(* CODESYS project codesys_code_execution_speedTests.export
   Author: Toni Kucic
   Version: 1.0
   Description: Cheatsheet for programming a PLC in IEC61131-3 Structured text. Contains usage of operators and common functions.
   Title: Plc Structured Text Cheatsheet
   CompiledLibraryCompatibilityVersion: CODESYS V3.5 SP16
   Company: TK Automation

Project tree, tasks and I/O mapping:
  CODESYS_Control_Win_V3_x64 : CODESYS Control Win V3 x64, 3S - Smart Software Solutions GmbH, version 3.5.18.20
    application Application
      libraries: MemoryUtils, 3.5.18.0 (3S - Smart Software Solutions GmbH)
      task Task (cyclic, interval 200 ms, priority 1) calls speedRunner
  CODESYS_Control_RTE_V3_x64 : CODESYS Control RTE V3 x64, 3S - Smart Software Solutions GmbH, version 3.5.18.20
    application Application
      libraries: MemoryUtils, 3.5.18.0 (3S - Smart Software Solutions GmbH)
      task Task (cyclic, interval 200 ms, priority 1) calls speedRunner
  libraries: Standard, 3.5.18.0 (System)
  01 - Impact of dynamic arrays/
    program x01_ImpactOfDynamicArrays [ST]
  02 - Execution speed of PLC languages/
    program x02_ExecSpeedOfLanguageTypes [ST]
    function addTwoIntsLadder [LD]
    function addTwoIntsST [ST]
    function addTwoIntsFBD [FBD]
  03 - Floating point operations/
    program x03_FloatingPointOperations [ST]
  04 - Function overhead/
    function addTwoInts [ST]
    program x04_FunctionOverhead [ST]: addTwoNumbers
  05 - MemSet over Data Zero/
    program x05_MemSetVsDataZeero [ST]
    data type dtTestStruct
  06 - SHL over MemCpy/
    program x06_ShlVsMemCpy [ST]
  07 - String operations/
    program x07_StringOperations [ST]
  08 - Operations with booleans/
    program x08_CheckingBools [ST]
  09 - Case versus IF ELSIF/
    program x09_CaseVsIfElsif [ST]: returnIndexIfElsif, returnIndexCase
  10 - Bit operations/
    program x10_1_BitAccess [ST]
    data type dtBitStruct
    program x10_3_BitMath [ST]
    program x10_2_BitSet [ST]
    function checkBit_bitmask [ST]
    function setBit_bitmask [ST]
    function clearBit_bitmask [ST]
    function setBitToValue_bitmask [ST]
    function setBit_dotNot [ST]
    function checkBit_dotNot [ST]
    function clearBit_dotNot [ST]
    function checkBit_bitStruct [ST]
    function clearBit_bitStruct [ST]
    function setBit_bitStruct [ST]
    function setBitToValue_bitStruct [ST]
    function setBitToValue_dotNot [ST]
  TestFramework/
    function calcAVG [ST]
    data type dtSpeedTest
    program speedRunner [ST]
*)

// 05 - MemSet over Data Zero/dtTestStruct
TYPE dtTestStruct :
STRUCT
	dummy1 : USINT := 255;
	Elem1 : INT := -1;
	Id : DWORD := 215215126;
	IdText : STRING := 'Testing for speed';
	dummy2 : ARRAY[0..11] OF DWORD;
	dummy4 : BOOL := FALSE;
	dummy5 : STRING[255] := 'Big array';
	dummy6 : LINT := 1211212723838939;
END_STRUCT
END_TYPE

// 10 - Bit operations/dtBitStruct
TYPE dtBitStruct :
STRUCT
	bit1 : BIT;
	bit2 : BIT;
	bit3 : BIT;
	bit4 : BIT;
	bit5 : BIT;
	bit6 : BIT;
	bit7 : BIT;
	bit8 : BIT;
	bit9 : BIT;
	bit10 : BIT;
	bit11 : BIT;
	bit12 : BIT;
	bit13 : BIT;
	bit14 : BIT;
	bit15 : BIT;
	bit16 : BIT;
END_STRUCT
END_TYPE

// TestFramework/dtSpeedTest
TYPE dtSpeedTest :
STRUCT
	Results 			: ARRAY[0..9] OF LTIME;
	AverageExecTime  	: LTIME;
	OldTime     		: LTIME;
	ExecTime    		: LTIME;
END_STRUCT
END_TYPE

// TestFramework/speedRunner
PROGRAM speedRunner
VAR
	vOldTime : LTIME;
	vTimeToRunTests : LTIME;
	vStart : BOOL := TRUE;
END_VAR

IF vStart THEN
	vOldTime := LTIME();
	vStart := FALSE;
END_IF

(*Run tests one by one*)
x01_ImpactOfDynamicArrays();
x02_ExecSpeedOfLanguageTypes();
x03_FloatingPointOperations();
x04_FunctionOverhead();
x05_MemSetVsDataZeero();
x06_ShlVsMemCpy();
x07_StringOperations();
x08_CheckingBools();
x09_CaseVsIfElsif();
x10_1_BitAccess();
x10_2_BitSet();
x10_3_BitMath();

IF x01_ImpactOfDynamicArrays.vRunDone
AND x02_ExecSpeedOfLanguageTypes.vRunDone
AND x03_FloatingPointOperations.vRunDone
AND x04_FunctionOverhead.vRunDone
AND x05_MemSetVsDataZeero.vRunDone
AND x06_ShlVsMemCpy.vRunDone
AND x07_StringOperations.vRunDone
AND x08_CheckingBools.vRunDone
AND x09_CaseVsIfElsif.vRunDone
AND x10_1_BitAccess.vRunDone
AND x10_2_BitSet.vRunDone
AND x10_3_BitMath.vRunDone
AND vTimeToRunTests = LTIME#0S
 THEN
	vTimeToRunTests := LTIME() - vOldTime;
END_IF

END_PROGRAM

// 01 - Impact of dynamic arrays/x01_ImpactOfDynamicArrays
PROGRAM x01_ImpactOfDynamicArrays
VAR CONSTANT
	cNrRuns : USINT(0..9) := 5;
	cRepeatCalcTimes : UDINT := 1000000; //1 Million times
END_VAR
VAR
	vRunsCompleted : USINT := 0;
	vRunDone : BOOL := FALSE;
	vTest1 : dtSpeedTest;
	vTest2 : dtSpeedTest;

	i : UDINT;
	
	//Test vars
	vAvgTimeFun : LTIME;
	vAvgTimeHardCoded : LTIME;
	vTimes : ARRAY[0..9] OF LTIME := [LTIME#1MS,LTIME#2MS,LTIME#3MS,LTIME#4MS,LTIME#5MS,LTIME#6MS,LTIME#7MS,LTIME#8MS,LTIME#9MS,LTIME#10MS];
	j : USINT;
END_VAR

IF vRunsCompleted > cNrRuns THEN
	vTest1.AverageExecTime := calcAvg(vTest1.Results);
	vTest2.AverageExecTime := calcAvg(vTest2.Results);
	vRunDone := TRUE;
	RETURN;
END_IF
	
//------------CALCULATION A -------------------
vTest1.OldTime := LTIME();
FOR i:= 0 TO cRepeatCalcTimes DO
	vAvgTimeFun := calcAvg(vTimes);
END_FOR
vTest1.ExecTime := LTIME() - vTest1.OldTime;

//------------CALCULATION B -------------------
vTest2.OldTime := LTIME();
FOR i:= 0 TO cRepeatCalcTimes DO
	vAvgTimeHardCoded := LTIME#0MS;
	FOR j:= 0 TO 9 DO
		vAvgTimeHardCoded := vAvgTimeHardCoded + vTimes[j];
	END_FOR
	vAvgTimeHardCoded := vAvgTimeHardCoded / j;
END_FOR
vTest2.ExecTime := LTIME() - vTest2.OldTime;

//------------CATCH RESULTS---------------------
vTest1.Results[vRunsCompleted] := vTest1.ExecTime;
vTest2.Results[vRunsCompleted] := vTest2.ExecTime;
vRunsCompleted := vRunsCompleted + 1;

END_PROGRAM

// TestFramework/calcAVG
FUNCTION calcAVG : LTIME
VAR_IN_OUT
	Results : ARRAY[*] OF LTIME;
END_VAR
VAR
	i : DINT;
END_VAR

FOR i:= LOWER_BOUND(Results,1) TO UPPER_BOUND(Results,1) DO
	calcAvg := calcAvg + Results[i];
END_FOR
calcAvg := calcAvg / i;
RETURN;

END_FUNCTION

// 02 - Execution speed of PLC languages/x02_ExecSpeedOfLanguageTypes
PROGRAM x02_ExecSpeedOfLanguageTypes
VAR CONSTANT
	cNrRuns : USINT(0..9) := 5;
	cRepeatCalcTimes : UDINT := 1000000; //1 Million times
END_VAR
VAR
	vRunsCompleted : USINT := 0;
	vRunDone : BOOL := FALSE;
	vTest1 : dtSpeedTest;
	vTest2 : dtSpeedTest;
	vTest3 : dtSpeedTest;
	i : UDINT;
	
	//Test vars
	vInt1 : INT := 1;
	vInt2 : INT := 2;
	vResult1 : INT;
	vResult2 : INT;
	vResult3 : INT;
END_VAR

IF vRunsCompleted > cNrRuns THEN
	vTest1.AverageExecTime := calcAvg(vTest1.Results); //User function Ladder
	vTest2.AverageExecTime := calcAvg(vTest2.Results); //User function ST
	vTest3.AverageExecTime := calcAvg(vTest3.Results); //User function FBD
	vRunDone := TRUE;
	RETURN;
END_IF
	
//------------CALCULATION A -------------------
vTest1.OldTime := LTIME();
FOR i:= 0 TO cRepeatCalcTimes DO
	vResult1 := addTwoIntsLadder(vInt1, vInt2);
END_FOR
vTest1.ExecTime := LTIME() - vTest1.OldTime;

//------------CALCULATION B -------------------
vTest2.OldTime := LTIME();
FOR i:= 0 TO cRepeatCalcTimes DO
	vResult2 := addTwoIntsST(vInt1, vInt2);
END_FOR
vTest2.ExecTime := LTIME() - vTest2.OldTime;

//------------CALCULATION C -------------------
vTest3.OldTime := LTIME();
FOR i:= 0 TO cRepeatCalcTimes DO
	vResult3 := addTwoIntsFBD(vInt1, vInt2);
END_FOR
vTest3.ExecTime := LTIME() - vTest3.OldTime;

//------------CATCH RESULTS---------------------
vTest1.Results[vRunsCompleted] := vTest1.ExecTime;
vTest2.Results[vRunsCompleted] := vTest2.ExecTime;
vTest3.Results[vRunsCompleted] := vTest3.ExecTime;
vRunsCompleted := vRunsCompleted + 1;

END_PROGRAM

// 02 - Execution speed of PLC languages/addTwoIntsLadder
FUNCTION addTwoIntsLadder : INT
VAR_INPUT
	Int1 : INT;
	Int2 : INT;
END_VAR
VAR
END_VAR

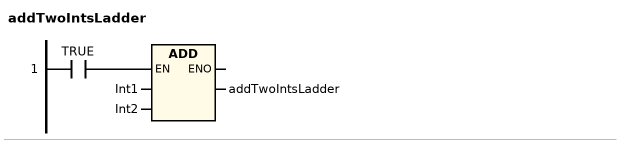
// NETWORK 1
addTwoIntsLadder := Int1 + Int2;

END_FUNCTION

// 02 - Execution speed of PLC languages/addTwoIntsST
FUNCTION addTwoIntsST : INT
VAR_INPUT
	int1 : INT;
	int2 : INT;
END_VAR
VAR
END_VAR

addTwoIntsST := int1 + int2;

END_FUNCTION

// 02 - Execution speed of PLC languages/addTwoIntsFBD
FUNCTION addTwoIntsFBD : INT
VAR_INPUT
	int1 : INT;
	int2 : INT;
END_VAR
VAR
END_VAR

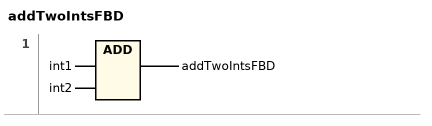
// NETWORK 1
addTwoIntsFBD := int1 + int2;

END_FUNCTION

// 03 - Floating point operations/x03_FloatingPointOperations
PROGRAM x03_FloatingPointOperations
VAR CONSTANT
	cNrRuns : USINT(0..9) := 5;
	cRepeatCalcTimes : UDINT := 1000000; //1 Million times
END_VAR
VAR
	vRunsCompleted : USINT := 0;
	vRunDone : BOOL := FALSE;
	vTest1 : dtSpeedTest;
	vTest2 : dtSpeedTest;
	vTest3 : dtSpeedTest;
	vTest4 : dtSpeedTest;
	vTest5 : dtSpeedTest;
	vTest6 : dtSpeedTest;
	vTest7 : dtSpeedTest;
	vTest8 : dtSpeedTest;
	vTest9 : dtSpeedTest;
	i : UDINT;
	
	//Test vars
	vInteger1 : INT := 1234;
	vInteger2 : INT := 4231;
	vReal1 : REAL := 1234.4231;
	vReal2 : REAL := 4231.1234;
	vInteger3 : DINT := 1234;
	vInteger4 : DINT := 4231;
	
	vResult1 : INT;
	vResult2 : REAL;
	vResult3 : DINT;
	vResult4 : INT;
	vResult5 : REAL;
	vResult6 : DINT;
	vResult7 : INT;
	vResult8 : REAL;
	vResult9 : DINT;
END_VAR

IF vRunsCompleted > cNrRuns THEN
	vTest1.AverageExecTime := calcAvg(vTest1.Results); //Time to add two integers 1 milion times
	vTest2.AverageExecTime := calcAvg(vTest2.Results); //Time to add two reals 1 milion times
	vTest3.AverageExecTime := calcAvg(vTest3.Results); //Time to add two DINTs (32b INT) 1 milion times
	vTest4.AverageExecTime := calcAvg(vTest4.Results); //Time to multiply two integers 1 milion times
	vTest5.AverageExecTime := calcAvg(vTest5.Results); //Time to multiply two reals 1 milion times
	vTest6.AverageExecTime := calcAvg(vTest6.Results); //Time to multiply two DINTs (32b INT) 1 milion times
	vTest7.AverageExecTime := calcAvg(vTest7.Results); //Time to divide two integers 1 milion times
	vTest8.AverageExecTime := calcAvg(vTest8.Results); //Time to divide two reals 1 milion times
	vTest9.AverageExecTime := calcAvg(vTest9.Results); //Time to divide two DINTs (32b INT) 1 milion times
	vRunDone := TRUE;	
	RETURN;
END_IF

//------------CALCULATION A -------------------
vTest1.OldTime := LTIME();
FOR i:= 0 TO cRepeatCalcTimes DO
	vResult1 := vInteger1 + vInteger2;
END_FOR
vTest1.ExecTime := LTIME() - vTest1.OldTime;

//------------CALCULATION B -------------------
vTest2.OldTime := LTIME();
FOR i:= 0 TO cRepeatCalcTimes DO
	vResult2 := vReal1 + vReal2;
END_FOR
vTest2.ExecTime := LTIME() - vTest2.OldTime;

//------------CALCULATION C -------------------
vTest3.OldTime := LTIME();
FOR i:= 0 TO cRepeatCalcTimes DO
	vResult3 := vInteger3 + vInteger4;
END_FOR
vTest3.ExecTime := LTIME() - vTest3.OldTime;

//------------CALCULATION D -------------------
vTest4.OldTime := LTIME();
FOR i:= 0 TO cRepeatCalcTimes DO
	vResult4 := vInteger1 * vInteger2;
END_FOR
vTest4.ExecTime := LTIME() - vTest4.OldTime;

//------------CALCULATION E -------------------
vTest5.OldTime := LTIME();
FOR i:= 0 TO cRepeatCalcTimes DO
	vResult5 := vReal1 * vReal2;
END_FOR
vTest5.ExecTime := LTIME() - vTest5.OldTime;

//------------CALCULATION F -------------------
vTest6.OldTime := LTIME();
FOR i:= 0 TO cRepeatCalcTimes DO
	vResult6 := vInteger3 * vInteger4;
END_FOR
vTest6.ExecTime := LTIME() - vTest6.OldTime;

//------------CALCULATION G -------------------
vTest7.OldTime := LTIME();
FOR i:= 0 TO cRepeatCalcTimes DO
	vResult7 := vInteger1 / vInteger2;
END_FOR
vTest7.ExecTime := LTIME() - vTest7.OldTime;

//------------CALCULATION H -------------------
vTest8.OldTime := LTIME();
FOR i:= 0 TO cRepeatCalcTimes DO
	vResult8 := vReal1 / vReal2;
END_FOR
vTest8.ExecTime := LTIME() - vTest8.OldTime;

//------------CALCULATION I -------------------
vTest9.OldTime := LTIME();
FOR i:= 0 TO cRepeatCalcTimes DO
	vResult9 := vInteger3 / vInteger4;
END_FOR
vTest9.ExecTime := LTIME() - vTest9.OldTime;


//------------CATCH RESULTS---------------------
vTest1.Results[vRunsCompleted] := vTest1.ExecTime;
vTest2.Results[vRunsCompleted] := vTest2.ExecTime;
vTest3.Results[vRunsCompleted] := vTest3.ExecTime;
vTest4.Results[vRunsCompleted] := vTest4.ExecTime;
vTest5.Results[vRunsCompleted] := vTest5.ExecTime;
vTest6.Results[vRunsCompleted] := vTest6.ExecTime;
vTest7.Results[vRunsCompleted] := vTest7.ExecTime;
vTest8.Results[vRunsCompleted] := vTest8.ExecTime;
vTest9.Results[vRunsCompleted] := vTest9.ExecTime;
vRunsCompleted := vRunsCompleted + 1;

END_PROGRAM

// 04 - Function overhead/x04_FunctionOverhead
PROGRAM x04_FunctionOverhead
VAR CONSTANT
	cNrRuns : USINT(0..9) := 5;
	cRepeatCalcTimes : UDINT := 1000000; //1 Million times
END_VAR
VAR
	vRunsCompleted : USINT := 0;
	vRunDone : BOOL := FALSE;
	vTest1 : dtSpeedTest;
	vTest2 : dtSpeedTest;
	vTest3 : dtSpeedTest;

	i : UDINT;
	
	//Test vars
	vInt1 : INT := 1;
	vInt2 : INT := 2;
	vResult1 : INT;
	vResult2 : INT;
	vResult3 : INT;
END_VAR

IF vRunsCompleted > cNrRuns THEN
	vTest1.AverageExecTime := calcAvg(vTest1.Results); //Operands
	vTest2.AverageExecTime := calcAvg(vTest2.Results); //User function
	vTest3.AverageExecTime := calcAvg(vTest3.Results); //PRG method
	vRunDone := TRUE;
	RETURN;
END_IF
	
//------------CALCULATION A -------------------
vTest1.OldTime := LTIME();
FOR i:= 0 TO cRepeatCalcTimes DO
	vResult1 := vInt1 + vInt2;
END_FOR
vTest1.ExecTime := LTIME() - vTest1.OldTime;

//------------CALCULATION B -------------------
vTest2.OldTime := LTIME();
FOR i:= 0 TO cRepeatCalcTimes DO
	vResult2 := addTwoInts(vInt1, vInt2);
END_FOR
vTest2.ExecTime := LTIME() - vTest2.OldTime;

//------------CALCULATION C -------------------
vTest3.OldTime := LTIME();
FOR i:= 0 TO cRepeatCalcTimes DO
	vResult3 := addTwoNumbers(vInt1, vInt2);
END_FOR
vTest3.ExecTime := LTIME() - vTest3.OldTime;

//------------CATCH RESULTS---------------------
vTest1.Results[vRunsCompleted] := vTest1.ExecTime;
vTest2.Results[vRunsCompleted] := vTest2.ExecTime;
vTest3.Results[vRunsCompleted] := vTest3.ExecTime;
vRunsCompleted := vRunsCompleted + 1;

METHOD PUBLIC addTwoNumbers : INT
VAR_INPUT
	int1 : INT;
	int2 : INT;
END_VAR
addTwoNumbers := int1 + int2;
END_METHOD

END_PROGRAM

// 04 - Function overhead/addTwoInts
FUNCTION addTwoInts : INT
VAR_IN_OUT
	int1 : INT;
	int2 : INT;
END_VAR
VAR
END_VAR

addTwoInts := int1 + int2;

END_FUNCTION

// 05 - MemSet over Data Zero/x05_MemSetVsDataZeero
PROGRAM x05_MemSetVsDataZeero
VAR CONSTANT
	cNrRuns : USINT(0..9) := 5;
	cRepeatCalcTimes : UDINT := 1000000; //1 Million times
	cEmptyStruct : dtTestStruct;
END_VAR
VAR
	vRunsCompleted : USINT := 0;
	vRunDone : BOOL := FALSE;
	vTest1 : dtSpeedTest;
	vTest2 : dtSpeedTest;

	i : UDINT;
	
	//Test variables
	vResultStruct1 : dtTestStruct;
	vResultStruct2 : dtTestStruct;
END_VAR

IF vRunsCompleted > cNrRuns THEN
	vTest1.AverageExecTime := calcAvg(vTest1.Results);
	vTest2.AverageExecTime := calcAvg(vTest2.Results);
	vRunDone := TRUE;
	RETURN;
END_IF
	
//------------CALCULATION A -------------------
vTest1.OldTime := LTIME();
FOR i:= 0 TO cRepeatCalcTimes DO
	//RESET STRUCT WITH A EMPTY STRUCT
	vResultStruct1 := cEmptyStruct;
END_FOR
vTest1.ExecTime := LTIME() - vTest1.OldTime;

//------------CALCULATION B -------------------
vTest2.OldTime := LTIME();
FOR i:= 0 TO cRepeatCalcTimes DO
	//RESET STRUCT WITH MEM SET
	MEMUtils.MemSet(pbyBuffer:= ADR(vResultStruct2), byValue:= 16#0 , dwSize:= SIZEOF(vResultStruct2));
END_FOR
vTest2.ExecTime := LTIME() - vTest2.OldTime;

//------------CATCH RESULTS---------------------
vTest1.Results[vRunsCompleted] := vTest1.ExecTime;
vTest2.Results[vRunsCompleted] := vTest2.ExecTime;
vRunsCompleted := vRunsCompleted + 1;

END_PROGRAM

// 06 - SHL over MemCpy/x06_ShlVsMemCpy
PROGRAM x06_ShlVsMemCpy
VAR CONSTANT
	cNrRuns : USINT(0..9) := 5;
	cRepeatCalcTimes : UDINT := 1000000; //1 Million times
END_VAR
VAR
	vRunsCompleted : USINT := 0;
	vRunDone : BOOL := FALSE;
	vTest1 : dtSpeedTest;
	vTest2 : dtSpeedTest;

	i : UDINT;
	
	//Test vars
	vSHRInteger : UINT;
	vMcpyInteger : UINT;
	vBuffer : ARRAY[0..1] OF USINT := [16#55, 16#AA];
	
	vSHLOldTime : LTIME;
	vMcpyOldTime : LTIME;
	
	vSHLExecTime : LTIME;
	vMcpyExecTime : LTIME;
	
END_VAR

IF vRunsCompleted > cNrRuns THEN
	vTest1.AverageExecTime := calcAvg(vTest1.Results);
	vTest2.AverageExecTime := calcAvg(vTest2.Results);
	vRunDone := TRUE;
	RETURN;
END_IF
	

vTest1.OldTime := LTIME();
FOR i:= 0 TO cRepeatCalcTimes DO
	//Assemble an UINT from two USINTs using SHR operator
	vSHRInteger := vBuffer[0] + SHL(vBuffer[1],8);
END_FOR
vTest1.ExecTime := LTIME() - vTest1.OldTime;

vTest2.OldTime := LTIME();
FOR i:= 0 TO cRepeatCalcTimes DO
	//Assemble an UINT from two USINTs using MemCpy
	MEMUtils.MemCpy(pbyDest:= ADR(vMcpyInteger), pbySrc:= ADR(vBuffer) , dwSize:= SIZEOF(vMcpyInteger));
END_FOR
vTest2.ExecTime := LTIME() - vTest2.OldTime;

//Results
vTest1.Results[vRunsCompleted] := vTest1.ExecTime;
vTest2.Results[vRunsCompleted] := vTest2.ExecTime;
vRunsCompleted := vRunsCompleted + 1;

END_PROGRAM

// 07 - String operations/x07_StringOperations
PROGRAM x07_StringOperations
VAR CONSTANT
	cNrRuns : USINT(0..9) := 5;
	cRepeatCalcTimes : UDINT := 1000000; //1 Million times
END_VAR
VAR
	vRunsCompleted : USINT := 0;
	vRunDone : BOOL := FALSE;
	vTest1 : dtSpeedTest;
	vTest2 : dtSpeedTest;
	vTest3 : dtSpeedTest;
	vTest4 : dtSpeedTest;
	vTest5 : dtSpeedTest;
	vTest6 : dtSpeedTest;
	i : UDINT;
	
	//Test vars
	vString1 : STRING[255] := 'Test string1';
	vString2 : STRING := 'Test string2';
	vString3 : STRING := 'a';
	vString4 : STRING := 'a';
	vByte :	BYTE := 16#FF;
	vArrByte :	ARRAY[0..255] OF BYTE;
	vResult1 : STRING[255];
	vResult2 : STRING;
	vResult3 : STRING;
	vResult4 : STRING[255];
	vResult5 : BYTE;
	vResult6 : ARRAY[0..255] OF BYTE;
	vSizes : ARRAY[0..3] OF UDINT;
END_VAR

IF vRunsCompleted > cNrRuns THEN
	vTest1.AverageExecTime := calcAvg(vTest1.Results); //Time to copy a string[255] 1 Million times
	vTest2.AverageExecTime := calcAvg(vTest2.Results); //Time to copy a string 1 Million times
	vTest3.AverageExecTime := calcAvg(vTest3.Results); //Time to concatenate 1 Million times characters with STRING
	vTest4.AverageExecTime := calcAvg(vTest4.Results); //Time to concatenate 1 Million times  characters with STRING[255]
	vTest5.AverageExecTime := calcAvg(vTest5.Results); //Time to move a byte 1 Million times
	vTest6.AverageExecTime := calcAvg(vTest6.Results); //Time to copy an array of 255 BYTE 1 Million times
	vRunDone := TRUE;
	RETURN;
END_IF

vSizes[0] := SIZEOF(vString1); //Size is 255 characters + zero char
vSizes[1] := SIZEOF(vString2); //Size is 80 characters + zero char, default if no size specified
vSizes[2] := SIZEOF(vResult3); //Size is 81, even though we concatenated 1 Million characters. The rest were chopped off
vSizes[3] := SIZEOF(vResult4); //Size is expected 256, other 744 characters chopped off

//------------CALCULATION A -------------------
vTest1.OldTime := LTIME();
FOR i:= 0 TO cRepeatCalcTimes DO
	vResult1 := vString1;
END_FOR
vTest1.ExecTime := LTIME() - vTest1.OldTime;

//------------CALCULATION B -------------------
vTest2.OldTime := LTIME();
FOR i:= 0 TO cRepeatCalcTimes DO
	vResult2 := vString2;
END_FOR
vTest2.ExecTime := LTIME() - vTest2.OldTime;

//------------CALCULATION C -------------------
vTest3.OldTime := LTIME();
FOR i:= 0 TO cRepeatCalcTimes DO
	vResult3 := CONCAT(vResult3, vString3);
END_FOR
vTest3.ExecTime := LTIME() - vTest3.OldTime;

//------------CALCULATION D -------------------
vTest4.OldTime := LTIME();
FOR i:= 0 TO cRepeatCalcTimes DO
	vResult4 := CONCAT(vResult4, vString4);
END_FOR
vTest4.ExecTime := LTIME() - vTest4.OldTime;

//------------CALCULATION E -------------------
vTest5.OldTime := LTIME();
FOR i:= 0 TO cRepeatCalcTimes DO
	vResult5 := vByte;
END_FOR
vTest5.ExecTime := LTIME() - vTest5.OldTime;

//------------CALCULATION F -------------------
vTest6.OldTime := LTIME();
FOR i:= 0 TO cRepeatCalcTimes DO
	vResult6 := vArrByte;
END_FOR
vTest6.ExecTime := LTIME() - vTest6.OldTime;

//------------CATCH RESULTS---------------------
vTest1.Results[vRunsCompleted] := vTest1.ExecTime;
vTest2.Results[vRunsCompleted] := vTest2.ExecTime;
vTest3.Results[vRunsCompleted] := vTest3.ExecTime;
vTest4.Results[vRunsCompleted] := vTest4.ExecTime;
vTest5.Results[vRunsCompleted] := vTest5.ExecTime;
vTest6.Results[vRunsCompleted] := vTest6.ExecTime;
vRunsCompleted := vRunsCompleted + 1;

END_PROGRAM

// 08 - Operations with booleans/x08_CheckingBools
PROGRAM x08_CheckingBools
VAR CONSTANT
	cNrRuns : USINT(0..9) := 5;
	cRepeatCalcTimes : UDINT := 1000000; //1 Million times
END_VAR
VAR
	vRunsCompleted : USINT := 0;
	vRunDone : BOOL := FALSE;
	vTest1 : dtSpeedTest;
	vTest2 : dtSpeedTest;
	vTest3 : dtSpeedTest;
	vTest4 : dtSpeedTest;
	vTest5 : dtSpeedTest;
	i : UDINT;
	
	//Test vars
	vBool : BOOL := TRUE;
	vResult : BOOL;
	vCounter : UINT := 0;
	vCastedUint : UINT;
END_VAR

IF vRunsCompleted > cNrRuns THEN
	vTest1.AverageExecTime := calcAvg(vTest1.Results); //Time to run IF vBool = TRUE THEN 1 Million times
	vTest2.AverageExecTime := calcAvg(vTest2.Results); //Time to run IF vBool THEN 1 Million times
	vTest3.AverageExecTime := calcAvg(vTest3.Results); //Time to increment a counter using if sentence 1 Million times
	vTest4.AverageExecTime := calcAvg(vTest4.Results); //Time to increment a counter using bool to UINT 1 Million times
	vTest5.AverageExecTime := calcAvg(vTest5.Results); //Time to cast a bool to UINT 1 Million times
	vRunDone := TRUE;
	RETURN;
END_IF

//------------CALCULATION A -------------------
vTest1.OldTime := LTIME();
//FOR i:= 0 TO cRepeatCalcTimes DO
	IF vBool = TRUE THEN
		vResult := vBool;
	END_IF
//END_FOR
vTest1.ExecTime := LTIME() - vTest1.OldTime;

//------------CALCULATION B -------------------
vTest2.OldTime := LTIME();
//FOR i:= 0 TO cRepeatCalcTimes DO
	IF vBool THEN
		vResult := vBool;
	END_IF
//END_FOR
vTest2.ExecTime := LTIME() - vTest2.OldTime;

//------------CALCULATION C -------------------
vTest3.OldTime := LTIME();
//FOR i:= 0 TO cRepeatCalcTimes DO
	IF vBool THEN
		vCounter := vCounter + 1;
	END_IF
//END_FOR
vTest3.ExecTime := LTIME() - vTest3.OldTime;

//------------CALCULATION D -------------------
vTest4.OldTime := LTIME();
//FOR i:= 0 TO cRepeatCalcTimes DO
	vCounter := vCounter + BOOL_TO_UINT(vBool);
//END_FOR
vTest4.ExecTime := LTIME() - vTest4.OldTime;

//------------CALCULATION D -------------------
vTest5.OldTime := LTIME();
//FOR i:= 0 TO cRepeatCalcTimes DO
	;vCastedUint := BOOL_TO_UINT(vBool);
//END_FOR
vTest5.ExecTime := LTIME() - vTest5.OldTime;

//------------CATCH RESULTS---------------------
vTest1.Results[vRunsCompleted] := vTest1.ExecTime;
vTest2.Results[vRunsCompleted] := vTest2.ExecTime;
vTest3.Results[vRunsCompleted] := vTest3.ExecTime;
vTest4.Results[vRunsCompleted] := vTest4.ExecTime;
vTest5.Results[vRunsCompleted] := vTest5.ExecTime;
vRunsCompleted := vRunsCompleted + 1;

END_PROGRAM

// 09 - Case versus IF ELSIF/x09_CaseVsIfElsif
PROGRAM x09_CaseVsIfElsif
VAR CONSTANT
	cNrRuns : USINT(0..9) := 5;
	cRepeatCalcTimes : UDINT := 1000000; //1 Million times
END_VAR
VAR
	vRunsCompleted : USINT := 0;
	vRunDone : BOOL := FALSE;
	vTest1 : dtSpeedTest;
	vTest2 : dtSpeedTest;
	vTest3 : dtSpeedTest;
	vTest4 : dtSpeedTest;
	vTest5 : dtSpeedTest;
	vTest6 : dtSpeedTest;
	i : UDINT;

	
	//Test vars
	vFirstIndex : INT := 15;
	vMiddleIndex : INT := 50;
	vLastIndex : INT := 99;
	
	vResultFirst : INT; //Should be 0
	vResultMiddle : INT; //Should be 50
	vResultLast : INT;//Should be 99

END_VAR

IF vRunsCompleted > cNrRuns THEN
	vTest1.AverageExecTime := calcAvg(vTest1.Results); //Time to run first branch of IF ELSIF 1 Million times
	vTest2.AverageExecTime := calcAvg(vTest2.Results); //Time to run middle branch of IF ELSIF 1 Million times
	vTest3.AverageExecTime := calcAvg(vTest3.Results); //Time to run last branch of IF ELSIF 1 Million times
	vTest4.AverageExecTime := calcAvg(vTest4.Results); //Time to run first branch of CASE 1 Million times
	vTest5.AverageExecTime := calcAvg(vTest5.Results); //Time to run middle branch of CASE 1 Million times
	vTest6.AverageExecTime := calcAvg(vTest6.Results); //Time to run last branch of CASE 1 Million times
	vRunDone := TRUE;
	RETURN;
END_IF

//------------CALCULATION A -------------------
vTest1.OldTime := LTIME();
FOR i:= 0 TO cRepeatCalcTimes DO
	vResultFirst := returnIndexIfElsif(vFirstIndex);
END_FOR
vTest1.ExecTime := LTIME() - vTest1.OldTime;

//------------CALCULATION B -------------------
vTest2.OldTime := LTIME();
FOR i:= 0 TO cRepeatCalcTimes DO
	vResultMiddle := returnIndexIfElsif(vMiddleIndex);
END_FOR
vTest2.ExecTime := LTIME() - vTest2.OldTime;

//------------CALCULATION C -------------------
vTest3.OldTime := LTIME();
FOR i:= 0 TO cRepeatCalcTimes DO
	vResultLast := returnIndexIfElsif(vLastIndex);
END_FOR
vTest3.ExecTime := LTIME() - vTest3.OldTime;

//------------CALCULATION D -------------------
vTest4.OldTime := LTIME();
FOR i:= 0 TO cRepeatCalcTimes DO
	vResultFirst := returnIndexCase(vFirstIndex);
END_FOR
vTest4.ExecTime := LTIME() - vTest4.OldTime;

//------------CALCULATION E -------------------
vTest5.OldTime := LTIME();
FOR i:= 0 TO cRepeatCalcTimes DO
	vResultMiddle := returnIndexCase(vMiddleIndex);
END_FOR
vTest5.ExecTime := LTIME() - vTest5.OldTime;

//------------CALCULATION F -------------------
vTest6.OldTime := LTIME();
FOR i:= 0 TO cRepeatCalcTimes DO
	vResultLast := returnIndexCase(vLastIndex);
END_FOR
vTest6.ExecTime := LTIME() - vTest6.OldTime;

//------------CATCH RESULTS---------------------
vTest1.Results[vRunsCompleted] := vTest1.ExecTime;
vTest2.Results[vRunsCompleted] := vTest2.ExecTime;
vTest3.Results[vRunsCompleted] := vTest3.ExecTime;
vTest4.Results[vRunsCompleted] := vTest4.ExecTime;
vTest5.Results[vRunsCompleted] := vTest5.ExecTime;
vTest6.Results[vRunsCompleted] := vTest6.ExecTime;

vRunsCompleted := vRunsCompleted + 1;

METHOD INTERNAL returnIndexIfElsif : INT
VAR_INPUT
	searchValue : INT;
END_VAR
IF searchValue = 0 THEN
        returnIndexIfElsif:=0;
        RETURN;

ELSIF searchValue = 1 THEN
        returnIndexIfElsif:= 1;
        RETURN;

ELSIF searchValue = 2 THEN
        returnIndexIfElsif:= 2;
        RETURN;

ELSIF searchValue = 3 THEN
        returnIndexIfElsif:= 3;
        RETURN;

ELSIF searchValue = 4 THEN
        returnIndexIfElsif:= 4;
        RETURN;

ELSIF searchValue = 5 THEN
        returnIndexIfElsif:= 5;
        RETURN;

ELSIF searchValue = 6 THEN
        returnIndexIfElsif:= 6;
        RETURN;

ELSIF searchValue = 7 THEN
        returnIndexIfElsif:= 7;
        RETURN;

ELSIF searchValue = 8 THEN
        returnIndexIfElsif:= 8;
        RETURN;

ELSIF searchValue = 9 THEN
        returnIndexIfElsif:= 9;
        RETURN;

ELSIF searchValue = 10 THEN
        returnIndexIfElsif:= 10;
        RETURN;

ELSIF searchValue = 11 THEN
        returnIndexIfElsif:= 11;
        RETURN;

ELSIF searchValue = 12 THEN
        returnIndexIfElsif:= 12;
        RETURN;

ELSIF searchValue = 13 THEN
        returnIndexIfElsif:= 13;
        RETURN;

ELSIF searchValue = 14 THEN
        returnIndexIfElsif:= 14;
        RETURN;

ELSIF searchValue = 15 THEN
        returnIndexIfElsif:= 15;
        RETURN;

ELSIF searchValue = 16 THEN
        returnIndexIfElsif:= 16;
        RETURN;

ELSIF searchValue = 17 THEN
        returnIndexIfElsif:= 17;
        RETURN;

ELSIF searchValue = 18 THEN
        returnIndexIfElsif:= 18;
        RETURN;

ELSIF searchValue = 19 THEN
        returnIndexIfElsif:= 19;
        RETURN;

ELSIF searchValue = 20 THEN
        returnIndexIfElsif:= 20;
        RETURN;

ELSIF searchValue = 21 THEN
        returnIndexIfElsif:= 21;
        RETURN;

ELSIF searchValue = 22 THEN
        returnIndexIfElsif:= 22;
        RETURN;

ELSIF searchValue = 23 THEN
        returnIndexIfElsif:= 23;
        RETURN;

ELSIF searchValue = 24 THEN
        returnIndexIfElsif:= 24;
        RETURN;

ELSIF searchValue = 25 THEN
        returnIndexIfElsif:= 25;
        RETURN;

ELSIF searchValue = 26 THEN
        returnIndexIfElsif:= 26;
        RETURN;

ELSIF searchValue = 27 THEN
        returnIndexIfElsif:= 27;
        RETURN;

ELSIF searchValue = 28 THEN
        returnIndexIfElsif:= 28;
        RETURN;

ELSIF searchValue = 29 THEN
        returnIndexIfElsif:= 29;
        RETURN;

ELSIF searchValue = 30 THEN
        returnIndexIfElsif:= 30;
        RETURN;

ELSIF searchValue = 31 THEN
        returnIndexIfElsif:= 31;
        RETURN;

ELSIF searchValue = 32 THEN
        returnIndexIfElsif:= 32;
        RETURN;

ELSIF searchValue = 33 THEN
        returnIndexIfElsif:= 33;
        RETURN;

ELSIF searchValue = 34 THEN
        returnIndexIfElsif:= 34;
        RETURN;

ELSIF searchValue = 35 THEN
        returnIndexIfElsif:= 35;
        RETURN;

ELSIF searchValue = 36 THEN
        returnIndexIfElsif:= 36;
        RETURN;

ELSIF searchValue = 37 THEN
        returnIndexIfElsif:= 37;
        RETURN;

ELSIF searchValue = 38 THEN
        returnIndexIfElsif:= 38;
        RETURN;

ELSIF searchValue = 39 THEN
        returnIndexIfElsif:= 39;
        RETURN;

ELSIF searchValue = 40 THEN
        returnIndexIfElsif:= 40;
        RETURN;

ELSIF searchValue = 41 THEN
        returnIndexIfElsif:= 41;
        RETURN;

ELSIF searchValue = 42 THEN
        returnIndexIfElsif:= 42;
        RETURN;

ELSIF searchValue = 43 THEN
        returnIndexIfElsif:= 43;
        RETURN;

ELSIF searchValue = 44 THEN
        returnIndexIfElsif:= 44;
        RETURN;

ELSIF searchValue = 45 THEN
        returnIndexIfElsif:= 45;
        RETURN;

ELSIF searchValue = 46 THEN
        returnIndexIfElsif:= 46;
        RETURN;

ELSIF searchValue = 47 THEN
        returnIndexIfElsif:= 47;
        RETURN;

ELSIF searchValue = 48 THEN
        returnIndexIfElsif:= 48;
        RETURN;

ELSIF searchValue = 49 THEN
        returnIndexIfElsif:= 49;
        RETURN;

ELSIF searchValue = 50 THEN
        returnIndexIfElsif:= 50;
        RETURN;

ELSIF searchValue = 51 THEN
        returnIndexIfElsif:= 51;
        RETURN;

ELSIF searchValue = 52 THEN
        returnIndexIfElsif:= 52;
        RETURN;

ELSIF searchValue = 53 THEN
        returnIndexIfElsif:= 53;
        RETURN;

ELSIF searchValue = 54 THEN
        returnIndexIfElsif:= 54;
        RETURN;

ELSIF searchValue = 55 THEN
        returnIndexIfElsif:= 55;
        RETURN;

ELSIF searchValue = 56 THEN
        returnIndexIfElsif:= 56;
        RETURN;

ELSIF searchValue = 57 THEN
        returnIndexIfElsif:= 57;
        RETURN;

ELSIF searchValue = 58 THEN
        returnIndexIfElsif:= 58;
        RETURN;

ELSIF searchValue = 59 THEN
        returnIndexIfElsif:= 59;
        RETURN;

ELSIF searchValue = 60 THEN
        returnIndexIfElsif:= 60;
        RETURN;

ELSIF searchValue = 61 THEN
        returnIndexIfElsif:= 61;
        RETURN;

ELSIF searchValue = 62 THEN
        returnIndexIfElsif:= 62;
        RETURN;

ELSIF searchValue = 63 THEN
        returnIndexIfElsif:= 63;
        RETURN;

ELSIF searchValue = 64 THEN
        returnIndexIfElsif:= 64;
        RETURN;

ELSIF searchValue = 65 THEN
        returnIndexIfElsif:= 65;
        RETURN;

ELSIF searchValue = 66 THEN
        returnIndexIfElsif:= 66;
        RETURN;

ELSIF searchValue = 67 THEN
        returnIndexIfElsif:= 67;
        RETURN;

ELSIF searchValue = 68 THEN
        returnIndexIfElsif:= 68;
        RETURN;

ELSIF searchValue = 69 THEN
        returnIndexIfElsif:= 69;
        RETURN;

ELSIF searchValue = 70 THEN
        returnIndexIfElsif:= 70;
        RETURN;

ELSIF searchValue = 71 THEN
        returnIndexIfElsif:= 71;
        RETURN;

ELSIF searchValue = 72 THEN
        returnIndexIfElsif:= 72;
        RETURN;

ELSIF searchValue = 73 THEN
        returnIndexIfElsif:= 73;
        RETURN;

ELSIF searchValue = 74 THEN
        returnIndexIfElsif:= 74;
        RETURN;

ELSIF searchValue = 75 THEN
        returnIndexIfElsif:= 75;
        RETURN;

ELSIF searchValue = 76 THEN
        returnIndexIfElsif:= 76;
        RETURN;

ELSIF searchValue = 77 THEN
        returnIndexIfElsif:= 77;
        RETURN;

ELSIF searchValue = 78 THEN
        returnIndexIfElsif:= 78;
        RETURN;

ELSIF searchValue = 79 THEN
        returnIndexIfElsif:= 79;
        RETURN;

ELSIF searchValue = 80 THEN
        returnIndexIfElsif:= 80;
        RETURN;

ELSIF searchValue = 81 THEN
        returnIndexIfElsif:= 81;
        RETURN;

ELSIF searchValue = 82 THEN
        returnIndexIfElsif:= 82;
        RETURN;

ELSIF searchValue = 83 THEN
        returnIndexIfElsif:= 83;
        RETURN;

ELSIF searchValue = 84 THEN
        returnIndexIfElsif:= 84;
        RETURN;

ELSIF searchValue = 85 THEN
        returnIndexIfElsif:= 85;
        RETURN;

ELSIF searchValue = 86 THEN
        returnIndexIfElsif:= 86;
        RETURN;

ELSIF searchValue = 87 THEN
        returnIndexIfElsif:= 87;
        RETURN;

ELSIF searchValue = 88 THEN
        returnIndexIfElsif:= 88;
        RETURN;

ELSIF searchValue = 89 THEN
        returnIndexIfElsif:= 89;
        RETURN;

ELSIF searchValue = 90 THEN
        returnIndexIfElsif:= 90;
        RETURN;

ELSIF searchValue = 91 THEN
        returnIndexIfElsif:= 91;
        RETURN;

ELSIF searchValue = 92 THEN
        returnIndexIfElsif:= 92;
        RETURN;

ELSIF searchValue = 93 THEN
        returnIndexIfElsif:= 93;
        RETURN;

ELSIF searchValue = 94 THEN
        returnIndexIfElsif:= 94;
        RETURN;

ELSIF searchValue = 95 THEN
        returnIndexIfElsif:= 95;
        RETURN;

ELSIF searchValue = 96 THEN
        returnIndexIfElsif:= 96;
        RETURN;

ELSIF searchValue = 97 THEN
        returnIndexIfElsif:= 97;
        RETURN;

ELSIF searchValue = 98 THEN
        returnIndexIfElsif:= 98;
        RETURN;

ELSIF searchValue = 99 THEN
        returnIndexIfElsif:= 99;
        RETURN;

END_IF
END_METHOD

METHOD INTERNAL returnIndexCase : INT
VAR_INPUT
	searchValue : INT;
END_VAR
CASE searchValue OF

        0: returnIndexCase := 0;
        RETURN;

        1: returnIndexCase := 1;
        RETURN;

        2: returnIndexCase := 2;
        RETURN;

        3: returnIndexCase := 3;
        RETURN;

        4: returnIndexCase := 4;
        RETURN;

        5: returnIndexCase := 5;
        RETURN;

        6: returnIndexCase := 6;
        RETURN;

        7: returnIndexCase := 7;
        RETURN;

        8: returnIndexCase := 8;
        RETURN;

        9: returnIndexCase := 9;
        RETURN;

        10: returnIndexCase := 10;
        RETURN;

        11: returnIndexCase := 11;
        RETURN;

        12: returnIndexCase := 12;
        RETURN;

        13: returnIndexCase := 13;
        RETURN;

        14: returnIndexCase := 14;
        RETURN;

        15: returnIndexCase := 15;
        RETURN;

        16: returnIndexCase := 16;
        RETURN;

        17: returnIndexCase := 17;
        RETURN;

        18: returnIndexCase := 18;
        RETURN;

        19: returnIndexCase := 19;
        RETURN;

        20: returnIndexCase := 20;
        RETURN;

        21: returnIndexCase := 21;
        RETURN;

        22: returnIndexCase := 22;
        RETURN;

        23: returnIndexCase := 23;
        RETURN;

        24: returnIndexCase := 24;
        RETURN;

        25: returnIndexCase := 25;
        RETURN;

        26: returnIndexCase := 26;
        RETURN;

        27: returnIndexCase := 27;
        RETURN;

        28: returnIndexCase := 28;
        RETURN;

        29: returnIndexCase := 29;
        RETURN;

        30: returnIndexCase := 30;
        RETURN;

        31: returnIndexCase := 31;
        RETURN;

        32: returnIndexCase := 32;
        RETURN;

        33: returnIndexCase := 33;
        RETURN;

        34: returnIndexCase := 34;
        RETURN;

        35: returnIndexCase := 35;
        RETURN;

        36: returnIndexCase := 36;
        RETURN;

        37: returnIndexCase := 37;
        RETURN;

        38: returnIndexCase := 38;
        RETURN;

        39: returnIndexCase := 39;
        RETURN;

        40: returnIndexCase := 40;
        RETURN;

        41: returnIndexCase := 41;
        RETURN;

        42: returnIndexCase := 42;
        RETURN;

        43: returnIndexCase := 43;
        RETURN;

        44: returnIndexCase := 44;
        RETURN;

        45: returnIndexCase := 45;
        RETURN;

        46: returnIndexCase := 46;
        RETURN;

        47: returnIndexCase := 47;
        RETURN;

        48: returnIndexCase := 48;
        RETURN;

        49: returnIndexCase := 49;
        RETURN;

        50: returnIndexCase := 50;
        RETURN;

        51: returnIndexCase := 51;
        RETURN;

        52: returnIndexCase := 52;
        RETURN;

        53: returnIndexCase := 53;
        RETURN;

        54: returnIndexCase := 54;
        RETURN;

        55: returnIndexCase := 55;
        RETURN;

        56: returnIndexCase := 56;
        RETURN;

        57: returnIndexCase := 57;
        RETURN;

        58: returnIndexCase := 58;
        RETURN;

        59: returnIndexCase := 59;
        RETURN;

        60: returnIndexCase := 60;
        RETURN;

        61: returnIndexCase := 61;
        RETURN;

        62: returnIndexCase := 62;
        RETURN;

        63: returnIndexCase := 63;
        RETURN;

        64: returnIndexCase := 64;
        RETURN;

        65: returnIndexCase := 65;
        RETURN;

        66: returnIndexCase := 66;
        RETURN;

        67: returnIndexCase := 67;
        RETURN;

        68: returnIndexCase := 68;
        RETURN;

        69: returnIndexCase := 69;
        RETURN;

        70: returnIndexCase := 70;
        RETURN;

        71: returnIndexCase := 71;
        RETURN;

        72: returnIndexCase := 72;
        RETURN;

        73: returnIndexCase := 73;
        RETURN;

        74: returnIndexCase := 74;
        RETURN;

        75: returnIndexCase := 75;
        RETURN;

        76: returnIndexCase := 76;
        RETURN;

        77: returnIndexCase := 77;
        RETURN;

        78: returnIndexCase := 78;
        RETURN;

        79: returnIndexCase := 79;
        RETURN;

        80: returnIndexCase := 80;
        RETURN;

        81: returnIndexCase := 81;
        RETURN;

        82: returnIndexCase := 82;
        RETURN;

        83: returnIndexCase := 83;
        RETURN;

        84: returnIndexCase := 84;
        RETURN;

        85: returnIndexCase := 85;
        RETURN;

        86: returnIndexCase := 86;
        RETURN;

        87: returnIndexCase := 87;
        RETURN;

        88: returnIndexCase := 88;
        RETURN;

        89: returnIndexCase := 89;
        RETURN;

        90: returnIndexCase := 90;
        RETURN;

        91: returnIndexCase := 91;
        RETURN;

        92: returnIndexCase := 92;
        RETURN;

        93: returnIndexCase := 93;
        RETURN;

        94: returnIndexCase := 94;
        RETURN;

        95: returnIndexCase := 95;
        RETURN;

        96: returnIndexCase := 96;
        RETURN;

        97: returnIndexCase := 97;
        RETURN;

        98: returnIndexCase := 98;
        RETURN;

        99: returnIndexCase := 99;
        RETURN;

END_CASE
END_METHOD

END_PROGRAM

// 10 - Bit operations/x10_1_BitAccess
PROGRAM x10_1_BitAccess
VAR CONSTANT
	cNrRuns : USINT(0..9) := 5;
	cRepeatCalcTimes : UDINT := 1000000; //1 Million times
END_VAR
VAR
	vRunsCompleted : USINT := 0;
	vRunDone : BOOL := FALSE;
	vTest1 : dtSpeedTest;
	vTest2 : dtSpeedTest;
	vTest3 : dtSpeedTest;
	i : UDINT;

	
	//Test vars
	vCodesysBits : dtBitStruct;
	vNormalInt : UINT := 16#5555;
	
	vResult1 : BOOL;
	vResult2 : BOOL;
	vResult3 : BOOL;
END_VAR

IF vRunsCompleted > cNrRuns THEN
	vTest1.AverageExecTime := calcAvg(vTest1.Results); //Time to access bit 3 1 Million times in codesys bit struct
	vTest2.AverageExecTime := calcAvg(vTest2.Results); //Time to access bit 3 1 Million times in normal integer using . notation
	vTest3.AverageExecTime := calcAvg(vTest3.Results); //Time to access bit 3 1 Million times in normal integer using bit masking
	vRunDone := TRUE;
	RETURN;
END_IF

//------------CALCULATION A -------------------
vTest1.OldTime := LTIME();
FOR i:= 0 TO cRepeatCalcTimes DO
	vResult1 := checkBit_bitStruct(vCodesysBits,2);
END_FOR
vTest1.ExecTime := LTIME() - vTest1.OldTime;

//------------CALCULATION B -------------------
vTest2.OldTime := LTIME();
FOR i:= 0 TO cRepeatCalcTimes DO
	vResult2 := checkBit_dotNot(vNormalInt,2);
END_FOR
vTest2.ExecTime := LTIME() - vTest2.OldTime;

//------------CALCULATION C -------------------
vTest3.OldTime := LTIME();
FOR i:= 0 TO cRepeatCalcTimes DO
	vResult3 := checkBit_bitmask(vNormalInt, 2);
END_FOR
vTest3.ExecTime := LTIME() - vTest3.OldTime;

//------------CATCH RESULTS---------------------
vTest1.Results[vRunsCompleted] := vTest1.ExecTime;
vTest2.Results[vRunsCompleted] := vTest2.ExecTime;
vTest3.Results[vRunsCompleted] := vTest3.ExecTime;

vRunsCompleted := vRunsCompleted + 1;

END_PROGRAM

// 10 - Bit operations/checkBit_bitStruct
FUNCTION checkBit_bitStruct : BOOL
VAR_INPUT
	bits : dtBitStruct;
	bitToCheck : USINT;
END_VAR

CASE bitToCheck OF
	0: checkBit_bitStruct := bits.bit1;
	1: checkBit_bitStruct := bits.bit2;
	2: checkBit_bitStruct := bits.bit3;
	3: checkBit_bitStruct := bits.bit4;
	4: checkBit_bitStruct := bits.bit5;
	5: checkBit_bitStruct := bits.bit6;
	6: checkBit_bitStruct := bits.bit7;
	7: checkBit_bitStruct := bits.bit8;
	8: checkBit_bitStruct := bits.bit9;
	9: checkBit_bitStruct := bits.bit10;
	10: checkBit_bitStruct := bits.bit11;
	11: checkBit_bitStruct := bits.bit12;
	12: checkBit_bitStruct := bits.bit13;
	13: checkBit_bitStruct := bits.bit14;
	14: checkBit_bitStruct := bits.bit15;
	15: checkBit_bitStruct := bits.bit16;
END_CASE

END_FUNCTION

// 10 - Bit operations/checkBit_dotNot
FUNCTION checkBit_dotNot : BOOL
VAR_INPUT
	bits : UINT;
	bitToCheck : USINT;
END_VAR
VAR
END_VAR

CASE bitToCheck OF
	0: checkBit_dotNot := bits.0;
	1: checkBit_dotNot := bits.1;
	2: checkBit_dotNot := bits.2;
	3: checkBit_dotNot := bits.3;
	4: checkBit_dotNot := bits.4;
	5: checkBit_dotNot := bits.5;
	6: checkBit_dotNot := bits.6;
	7: checkBit_dotNot := bits.7;
	8: checkBit_dotNot := bits.8;
	9: checkBit_dotNot := bits.9;
	10: checkBit_dotNot := bits.10;
	11: checkBit_dotNot := bits.11;
	12: checkBit_dotNot := bits.12;
	13: checkBit_dotNot := bits.13;
	14: checkBit_dotNot := bits.14;
	15: checkBit_dotNot := bits.15;
END_CASE

END_FUNCTION

// 10 - Bit operations/checkBit_bitmask
FUNCTION checkBit_bitmask : BOOL
VAR_INPUT
	bits : UINT;
	bitToCheck : USINT;
END_VAR
VAR
END_VAR

checkBit_bitmask := (bits AND SHL(1, bitToCheck)) <> 0;

END_FUNCTION

// 10 - Bit operations/x10_2_BitSet
PROGRAM x10_2_BitSet
VAR CONSTANT
	cNrRuns : USINT(0..9) := 5;
	cRepeatCalcTimes : UDINT := 1000000; //1 Million times
END_VAR
VAR
	vRunsCompleted : USINT := 0;
	vRunDone : BOOL := FALSE;
	vTest1 : dtSpeedTest;
	vTest2 : dtSpeedTest;
	vTest3 : dtSpeedTest;
	i : UDINT;
	
	//Test vars
	vCodesysBits : dtBitStruct;
	vNormalInt : UINT := 16#0;
	vNormalInt2 : UINT := 16#0;
	vNormalInt3 : UINT := 16#0;
	vResult1 : BOOL;
	vResult2 : BOOL;
	vResult3 : BOOL;
	
END_VAR

IF vRunsCompleted > cNrRuns THEN
	vTest1.AverageExecTime := calcAvg(vTest1.Results); //Time to set bit 3 1 Million times in codesys bit struct
	vTest2.AverageExecTime := calcAvg(vTest2.Results); //Time to set bit 3 1 Million times in normal integer using . notation
	vTest3.AverageExecTime := calcAvg(vTest3.Results); //Time to set bit 3 1 Million times in normal integer using bit masking
	vRunDone := TRUE;
	RETURN;
END_IF

//------------CALCULATION A -------------------
vTest1.OldTime := LTIME();
FOR i:= 0 TO cRepeatCalcTimes DO
	setBit_bitStruct(vCodesysBits, 2);
END_FOR
vTest1.ExecTime := LTIME() - vTest1.OldTime;

//------------CALCULATION B -------------------
vTest2.OldTime := LTIME();
FOR i:= 0 TO cRepeatCalcTimes DO
	setBit_dotNot(vNormalInt, 2);
END_FOR
vTest2.ExecTime := LTIME() - vTest2.OldTime;

//------------CALCULATION C -------------------
vTest3.OldTime := LTIME();
FOR i:= 0 TO cRepeatCalcTimes DO
	setBit_bitmask(vNormalInt2, 2);
END_FOR
vTest3.ExecTime := LTIME() - vTest3.OldTime;

//------------CATCH RESULTS---------------------
vTest1.Results[vRunsCompleted] := vTest1.ExecTime;
vTest2.Results[vRunsCompleted] := vTest2.ExecTime;
vTest3.Results[vRunsCompleted] := vTest3.ExecTime;

vRunsCompleted := vRunsCompleted + 1;

END_PROGRAM

// 10 - Bit operations/setBit_bitStruct
FUNCTION setBit_bitStruct : BOOL
VAR_IN_OUT
	bits : dtBitStruct;
END_VAR
VAR_INPUT
	bitToSet : USINT;
END_VAR

CASE bitToSet OF
	0: bits.bit1 := TRUE;
	1: bits.bit2 := TRUE;
	2: bits.bit3 := TRUE;
	3: bits.bit4 := TRUE;
	4: bits.bit5 := TRUE;
	5: bits.bit6 := TRUE;
	6: bits.bit7 := TRUE;
	7: bits.bit8 := TRUE;
	8: bits.bit9 := TRUE;
	9: bits.bit10 := TRUE;
	10: bits.bit11 := TRUE;
	11: bits.bit12 := TRUE;
	12: bits.bit13 := TRUE;
	13: bits.bit14 := TRUE;
	14: bits.bit15 := TRUE;
	15: bits.bit16 := TRUE;
END_CASE

END_FUNCTION

// 10 - Bit operations/setBit_dotNot
FUNCTION setBit_dotNot : BOOL
VAR_IN_OUT
	bits : UINT;
END_VAR
VAR_INPUT
	bitToSet : USINT;
END_VAR

CASE bitToSet OF
	0: bits.0 := TRUE;
	1: bits.1 := TRUE;
	2: bits.2 := TRUE;
	3: bits.3 := TRUE;
	4: bits.4 := TRUE;
	5: bits.5 := TRUE;
	6: bits.6 := TRUE;
	7: bits.7 := TRUE;
	8: bits.8 := TRUE;
	9: bits.9 := TRUE;
	10: bits.10 := TRUE;
	11: bits.11 := TRUE;
	12: bits.12 := TRUE;
	13: bits.13 := TRUE;
	14: bits.14 := TRUE;
	15: bits.15 := TRUE;
END_CASE

END_FUNCTION

// 10 - Bit operations/setBit_bitmask
FUNCTION setBit_bitmask : BOOL
VAR_IN_OUT
	bits : UINT;
END_VAR
VAR_INPUT
	bitToSet : USINT;
END_VAR

bits := bits OR SHL(UINT#1, bitToSet);

END_FUNCTION

// 10 - Bit operations/x10_3_BitMath
PROGRAM x10_3_BitMath
VAR CONSTANT
	cNrRuns : USINT(0..9) := 5;
	cRepeatCalcTimes : UDINT := 1000000; //1 Million times
END_VAR
VAR
	vRunsCompleted : USINT := 0;
	vRunDone : BOOL := FALSE;
	vTest1 : dtSpeedTest;
	vTest2 : dtSpeedTest;
	vTest3 : dtSpeedTest;

	i : UDINT;
	
	//Test vars
	vCodesysBits : dtBitStruct := (bit1:=TRUE, bit2:=TRUE, bit3 := FALSE);
	vNormalInt : UINT := 2#11;
	vNormalInt2 : UINT := 2#11;
	vNormalInt3 : UINT := 2#11;
	
END_VAR

IF vRunsCompleted > cNrRuns THEN
	vTest1.AverageExecTime := calcAvg(vTest1.Results); //Time to and two bits and save it to another bit 1 Million times using codesys bit struct
	vTest2.AverageExecTime := calcAvg(vTest2.Results); //Time to and two bits and save it to another bit 1 Million times using . notation
	vTest3.AverageExecTime := calcAvg(vTest3.Results); //Time to and two bits and save it to another bit 1 Million times using bit masking
	vRunDone := TRUE;
	RETURN;
END_IF

//------------CALCULATION A -------------------
vTest1.OldTime := LTIME();
FOR i:= 0 TO cRepeatCalcTimes DO
	setBitToValue_bitStruct(vCodesysBits, 2, checkBit_bitStruct(vCodesysBits, 0) AND checkBit_bitStruct(vCodesysBits, 1));
END_FOR
vTest1.ExecTime := LTIME() - vTest1.OldTime;

//------------CALCULATION B -------------------
vTest2.OldTime := LTIME();
FOR i:= 0 TO cRepeatCalcTimes DO
	setBitToValue_dotNot(vNormalInt, 2, checkBit_dotNot(vNormalInt, 0) AND checkBit_dotNot(vNormalInt, 1));
END_FOR
vTest2.ExecTime := LTIME() - vTest2.OldTime;

//------------CALCULATION C -------------------
vTest3.OldTime := LTIME();
FOR i:= 0 TO cRepeatCalcTimes DO
	setBitTovalue_bitmask(vNormalInt2, 2, checkBit_bitmask(vNormalInt2, 0) AND checkBit_bitmask(vNormalInt2, 1));
END_FOR
vTest3.ExecTime := LTIME() - vTest3.OldTime;


//------------CATCH RESULTS---------------------
vTest1.Results[vRunsCompleted] := vTest1.ExecTime;
vTest2.Results[vRunsCompleted] := vTest2.ExecTime;
vTest3.Results[vRunsCompleted] := vTest3.ExecTime;

vRunsCompleted := vRunsCompleted + 1;

END_PROGRAM

// 10 - Bit operations/setBitToValue_bitStruct
FUNCTION setBitToValue_bitStruct : BOOL
VAR_IN_OUT
	bits : dtBitStruct;
END_VAR
VAR_INPUT
	bitToSet : USINT;
	value : BOOL;
END_VAR

IF value THEN
	setBit_bitStruct(bits, bitToSet);
ELSE
	clearBit_bitStruct(bits, bitToSet);
END_IF

END_FUNCTION

// 10 - Bit operations/clearBit_bitStruct
FUNCTION clearBit_bitStruct : BOOL
VAR_IN_OUT
	bits : dtBitStruct;
END_VAR
VAR_INPUT
	bitToClear : USINT;
END_VAR

CASE bitToClear OF
	0: bits.bit1 := FALSE;
	1: bits.bit2 := FALSE;
	2: bits.bit3 := FALSE;
	3: bits.bit4 := FALSE;
	4: bits.bit5 := FALSE;
	5: bits.bit6 := FALSE;
	6: bits.bit7 := FALSE;
	7: bits.bit8 := FALSE;
	8: bits.bit9 := FALSE;
	9: bits.bit10 := FALSE;
	10: bits.bit11 := FALSE;
	11: bits.bit12 := FALSE;
	12: bits.bit13 := FALSE;
	13: bits.bit14 := FALSE;
	14: bits.bit15 := FALSE;
	15: bits.bit16 := FALSE;
END_CASE

END_FUNCTION

// 10 - Bit operations/setBitToValue_dotNot
FUNCTION setBitToValue_dotNot : BOOL
VAR_IN_OUT
	bits : UINT;
END_VAR
VAR_INPUT
	bitToSet : USINT;
	value : BOOL;
END_VAR

IF value THEN
	setBit_dotNot(bits, bitToSet);
ELSE
	clearBit_dotNot(bits, bitToSet);
END_IF

END_FUNCTION

// 10 - Bit operations/clearBit_dotNot
FUNCTION clearBit_dotNot : BOOL
VAR_IN_OUT
	bits : UINT;
END_VAR
VAR_INPUT
	bitToClear : USINT;
END_VAR

CASE bitToClear OF
	0: bits.0 := FALSE;
	1: bits.1 := FALSE;
	2: bits.2 := FALSE;
	3: bits.3 := FALSE;
	4: bits.4 := FALSE;
	5: bits.5 := FALSE;
	6: bits.6 := FALSE;
	7: bits.7 := FALSE;
	8: bits.8 := FALSE;
	9: bits.9 := FALSE;
	10: bits.10 := FALSE;
	11: bits.11 := FALSE;
	12: bits.12 := FALSE;
	13: bits.13 := FALSE;
	14: bits.14 := FALSE;
	15: bits.15 := FALSE;
END_CASE

END_FUNCTION

// 10 - Bit operations/setBitToValue_bitmask
FUNCTION setBitToValue_bitmask : BOOL
VAR_IN_OUT
	bits : UINT;
END_VAR
VAR_INPUT
	bitToSet : USINT;
	value : BOOL;
END_VAR

IF value THEN
	setBit_bitmask(bits, bitToSet);
ELSE
	clearBit_bitmask(bits, bitToSet);
END_IF

END_FUNCTION

// 10 - Bit operations/clearBit_bitmask
FUNCTION clearBit_bitmask : BOOL
VAR_IN_OUT
	bits : UINT;
END_VAR
VAR_INPUT
	bitToClear : USINT;
END_VAR

bits := bits AND NOT SHL(UINT#1, bitToClear-1);

END_FUNCTION
